// TwinCAT 3 PLC project main
// ProgramVersion: 3.1.4024.0
// libraries:
//   Tc2_Standard, * (Beckhoff Automation GmbH)
//   Tc2_System, * (Beckhoff Automation GmbH)
//   Tc3_Module, * (Beckhoff Automation GmbH)
// project tree:
//   / GlobalTextList.TcGTLO, PlcTask.TcTTO, Visualization Manager.TcVMO (not stored)
//   POUs/ MAIN.TcPOU
//   VISUs/ Visu.TcVIS
// real-time tasks:
//   TASK PlcTask: cycle T#10ms, priority 20, ADS port 350

CONFIGURATION main
    RESOURCE PLC ON TwinCAT3
        TASK PlcTask(INTERVAL := T#10ms, PRIORITY := 20);
        PROGRAM MAIN WITH PlcTask : MAIN;
    END_RESOURCE
END_CONFIGURATION

// ---- POUs/MAIN.TcPOU
PROGRAM MAIN
VAR
	bKnop1: BOOL;
    bKnop2: BOOL;
    bKnop3: BOOL;
    bKnop4: BOOL;
    bKnop5: BOOL;
    bKnop6: BOOL;
	
	bLamp : BOOL;
	out: TOF;
END_VAR

//https://infosys.beckhoff.com/english.php?content=../content/1033/tcplclib_tc2_standard/74405003.html&id=

//In een appartementsgebouw staan in de traphal op de verschillende verdiepingen in totaal 6 drukknoppen.
//Als men één van de drukknoppen bedient gaat de verlichting branden.
//De verlichting blijft 3MIN. branden - tijdens de test gebruikt men 3S - vooraleer deze vanzelf uitschakelt.
//Bij iedere bediening van een drukknop zal de tijd terug beginnen te lopen vanaf 0 en blijven de lampen branden tot de ingestelde tijd is afgelopen.

out(IN:= bKnop1 OR bKnop2 OR bKnop3 OR bKnop4 OR bKnop5 OR bKnop6 , PT:= T#3S , Q=>bLamp , ET=> );

END_PROGRAM

// ---- GlobalTextList.TcGTLO
TEXTLIST GlobalTextList
  564 = 'Knop 1'
  833 = 'Knop 2'
  232 = 'Knop 3'
  425 = 'Knop 4'
  499 = 'Knop 5'
  214 = 'Knop 6'
  817 = 'Label'
END_TEXTLIST

// ---- VISUs/Visu.TcVIS
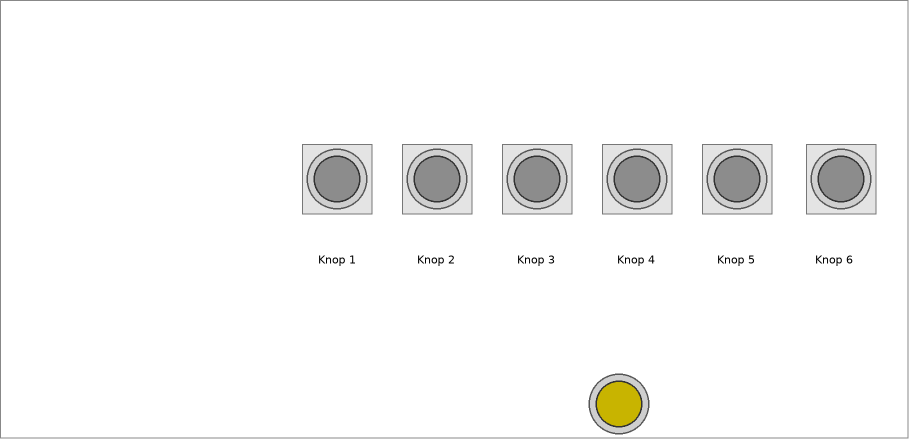
VISUALIZATION Visu  // 909x439
    PushSwitch (302,144 70x70), variable: MAIN.bKnop1, behaviour: TAP, style: Switch-PushSwitch-Gray
    PushSwitch (402,144 70x70), variable: MAIN.bKnop2, behaviour: TAP, style: Switch-PushSwitch-Gray
    PushSwitch (502,144 70x70), variable: MAIN.bKnop3, behaviour: TAP, style: Switch-PushSwitch-Gray
    PushSwitch (602,144 70x70), variable: MAIN.bKnop4, behaviour: TAP, style: Switch-PushSwitch-Gray
    PushSwitch (806,144 70x70), variable: MAIN.bKnop6, behaviour: TAP, style: Switch-PushSwitch-Gray
    PushSwitch (702,144 70x70), variable: MAIN.bKnop5, behaviour: TAP, style: Switch-PushSwitch-Gray
    Label (262,245 150x30), "Knop 1"
    Label (361,245 150x30), "Knop 2"
    Label (461,245 150x30), "Knop 3"
    Label (561,245 150x30), "Knop 4"
    Label (661,245 150x30), "Knop 5"
    Label (759,245 150x30), "Knop 6"
    Lamp1 (584,369 70x70), variable: MAIN.bLamp, style: Lamp-Lamp1-Yellow
END_VISUALIZATION
